// TIA Portal V16 export
// export: Created 2025-12-18T09:29:12.9038693Z, ExportSetting WithDefaults, DisplayName Totally Integrated Automation Portal, DisplayVersion V16, DisplayName TIA Portal Version Control Interface, DisplayVersion V16, DisplayName TIA Portal Openness, DisplayVersion V16, DisplayName STEP 7 Professional, DisplayVersion V16, DisplayName STEP 7 Safety, DisplayVersion V16, DisplayName WinCC Advanced, DisplayVersion V16
ORGANIZATION_BLOCK "Main"   // OB1, LAD, ProgramCycle
TITLE = "Main Program Sweep (Cycle)"
{ S7_Optimized_Access := 'TRUE' }
VERSION : 0.1
// stored: AutoNumber true, IsIECCheckEnabled false, SetENOAutomatically false
   VAR_INPUT
      Initial_Call : Bool;   // Initial call of this OB
      Remanence : Bool;   // =True, if remanent data are available
   END_VAR
   VAR_TEMP   // added for the SCL form of the ladder/FBD networks
      _w1 : Bool;
   END_VAR
BEGIN

REGION Network 1
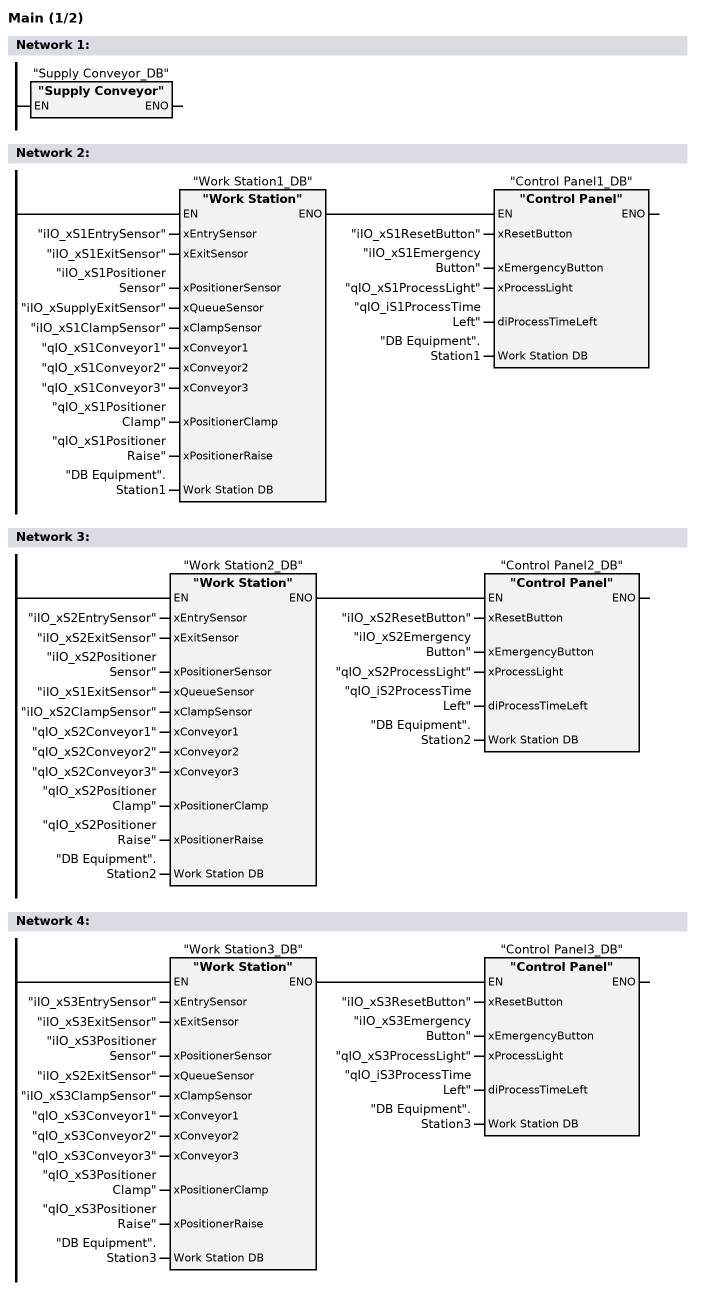
   RUNG wire#powerrail
      "Supply Conveyor_DB"()
   END_RUNG
   // the same network as SCL:
   "Supply Conveyor_DB"();   // "Supply Conveyor"
END_REGION

REGION Network 2
   RUNG wire#powerrail
      "Work Station1_DB"(xEntrySensor := "iIO_xS1EntrySensor", xExitSensor := "iIO_xS1ExitSensor", xPositionerSensor := "iIO_xS1PositionerSensor", xQueueSensor := "iIO_xSupplyExitSensor", xClampSensor := "iIO_xS1ClampSensor", xConveyor1 := "qIO_xS1Conveyor1", xConveyor2 := "qIO_xS1Conveyor2", xConveyor3 := "qIO_xS1Conveyor3", xPositionerClamp := "qIO_xS1PositionerClamp", xPositionerRaise := "qIO_xS1PositionerRaise", "Work Station DB" := "DB Equipment".Station1)
      "Control Panel1_DB"(xResetButton := "iIO_xS1ResetButton", xEmergencyButton := "iIO_xS1EmergencyButton", xProcessLight := "qIO_xS1ProcessLight", diProcessTimeLeft := "qIO_iS1ProcessTimeLeft", "Work Station DB" := "DB Equipment".Station1)
   END_RUNG
   // the same network as SCL:
   "Work Station1_DB"(xEntrySensor := "iIO_xS1EntrySensor",   // "Work Station"
                      xExitSensor := "iIO_xS1ExitSensor",
                      xPositionerSensor := "iIO_xS1PositionerSensor",
                      xQueueSensor := "iIO_xSupplyExitSensor",
                      xClampSensor := "iIO_xS1ClampSensor",
                      xConveyor1 := "qIO_xS1Conveyor1",
                      xConveyor2 := "qIO_xS1Conveyor2",
                      xConveyor3 := "qIO_xS1Conveyor3",
                      xPositionerClamp := "qIO_xS1PositionerClamp",
                      xPositionerRaise := "qIO_xS1PositionerRaise",
                      "Work Station DB" := "DB Equipment".Station1,
                      ENO => #_w1);
   IF #_w1 THEN
       "Control Panel1_DB"(xResetButton := "iIO_xS1ResetButton",   // "Control Panel"
                           xEmergencyButton := "iIO_xS1EmergencyButton",
                           xProcessLight := "qIO_xS1ProcessLight",
                           diProcessTimeLeft := "qIO_iS1ProcessTimeLeft",
                           "Work Station DB" := "DB Equipment".Station1);
   END_IF;
END_REGION

REGION Network 3
   RUNG wire#powerrail
      "Work Station2_DB"(xEntrySensor := "iIO_xS2EntrySensor", xExitSensor := "iIO_xS2ExitSensor", xPositionerSensor := "iIO_xS2PositionerSensor", xQueueSensor := "iIO_xS1ExitSensor", xClampSensor := "iIO_xS2ClampSensor", xConveyor1 := "qIO_xS2Conveyor1", xConveyor2 := "qIO_xS2Conveyor2", xConveyor3 := "qIO_xS2Conveyor3", xPositionerClamp := "qIO_xS2PositionerClamp", xPositionerRaise := "qIO_xS2PositionerRaise", "Work Station DB" := "DB Equipment".Station2)
      "Control Panel2_DB"(xResetButton := "iIO_xS2ResetButton", xEmergencyButton := "iIO_xS2EmergencyButton", xProcessLight := "qIO_xS2ProcessLight", diProcessTimeLeft := "qIO_iS2ProcessTimeLeft", "Work Station DB" := "DB Equipment".Station2)
   END_RUNG
   // the same network as SCL:
   "Work Station2_DB"(xEntrySensor := "iIO_xS2EntrySensor",   // "Work Station"
                      xExitSensor := "iIO_xS2ExitSensor",
                      xPositionerSensor := "iIO_xS2PositionerSensor",
                      xQueueSensor := "iIO_xS1ExitSensor",
                      xClampSensor := "iIO_xS2ClampSensor",
                      xConveyor1 := "qIO_xS2Conveyor1",
                      xConveyor2 := "qIO_xS2Conveyor2",
                      xConveyor3 := "qIO_xS2Conveyor3",
                      xPositionerClamp := "qIO_xS2PositionerClamp",
                      xPositionerRaise := "qIO_xS2PositionerRaise",
                      "Work Station DB" := "DB Equipment".Station2,
                      ENO => #_w1);
   IF #_w1 THEN
       "Control Panel2_DB"(xResetButton := "iIO_xS2ResetButton",   // "Control Panel"
                           xEmergencyButton := "iIO_xS2EmergencyButton",
                           xProcessLight := "qIO_xS2ProcessLight",
                           diProcessTimeLeft := "qIO_iS2ProcessTimeLeft",
                           "Work Station DB" := "DB Equipment".Station2);
   END_IF;
END_REGION

REGION Network 4
   RUNG wire#powerrail
      "Work Station3_DB"(xEntrySensor := "iIO_xS3EntrySensor", xExitSensor := "iIO_xS3ExitSensor", xPositionerSensor := "iIO_xS3PositionerSensor", xQueueSensor := "iIO_xS2ExitSensor", xClampSensor := "iIO_xS3ClampSensor", xConveyor1 := "qIO_xS3Conveyor1", xConveyor2 := "qIO_xS3Conveyor2", xConveyor3 := "qIO_xS3Conveyor3", xPositionerClamp := "qIO_xS3PositionerClamp", xPositionerRaise := "qIO_xS3PositionerRaise", "Work Station DB" := "DB Equipment".Station3)
      "Control Panel3_DB"(xResetButton := "iIO_xS3ResetButton", xEmergencyButton := "iIO_xS3EmergencyButton", xProcessLight := "qIO_xS3ProcessLight", diProcessTimeLeft := "qIO_iS3ProcessTimeLeft", "Work Station DB" := "DB Equipment".Station3)
   END_RUNG
   // the same network as SCL:
   "Work Station3_DB"(xEntrySensor := "iIO_xS3EntrySensor",   // "Work Station"
                      xExitSensor := "iIO_xS3ExitSensor",
                      xPositionerSensor := "iIO_xS3PositionerSensor",
                      xQueueSensor := "iIO_xS2ExitSensor",
                      xClampSensor := "iIO_xS3ClampSensor",
                      xConveyor1 := "qIO_xS3Conveyor1",
                      xConveyor2 := "qIO_xS3Conveyor2",
                      xConveyor3 := "qIO_xS3Conveyor3",
                      xPositionerClamp := "qIO_xS3PositionerClamp",
                      xPositionerRaise := "qIO_xS3PositionerRaise",
                      "Work Station DB" := "DB Equipment".Station3,
                      ENO => #_w1);
   IF #_w1 THEN
       "Control Panel3_DB"(xResetButton := "iIO_xS3ResetButton",   // "Control Panel"
                           xEmergencyButton := "iIO_xS3EmergencyButton",
                           xProcessLight := "qIO_xS3ProcessLight",
                           diProcessTimeLeft := "qIO_iS3ProcessTimeLeft",
                           "Work Station DB" := "DB Equipment".Station3);
   END_IF;
END_REGION

REGION Network 5
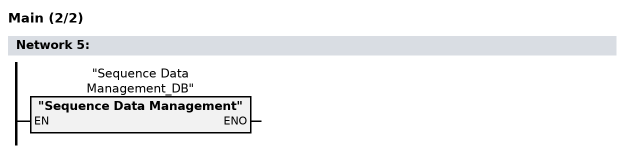
   RUNG wire#powerrail
      "Sequence Data Management_DB"()
   END_RUNG
   // the same network as SCL:
   "Sequence Data Management_DB"();   // "Sequence Data Management"
END_REGION
END_ORGANIZATION_BLOCK
